TYPE csp_case_glue_ls_accU_upperPosition_enum :
(
	CSP_CASE_GLUE_LS_ACCU_UPPERPOSITION_STATUS_NOT_INITIALIZED 									:= 0,
	CSP_CASE_GLUE_LS_ACCU_UPPERPOSITION_STATUS_DISABLED 										:= 10,
	CSP_CASE_GLUE_LS_ACCU_UPPERPOSITION_STATUS_POSITION_CHECK									:= 20,
	CSP_CASE_GLUE_LS_ACCU_UPPERPOSITION_STATUS_ENABLE_REQUEST 									:= 30,
	CSP_CASE_GLUE_LS_ACCU_UPPERPOSITION_STATUS_ENABLED 											:= 40,
	CSP_CASE_GLUE_LS_ACCU_UPPERPOSITION_STATUS_ABS_MOVE_REQUEST									:= 50,
	CSP_CASE_GLUE_LS_ACCU_UPPERPOSITION_STATUS_ABS_MOVING										:= 60,
	CSP_CASE_GLUE_LS_ACCU_UPPERPOSITION_STATUS_STOP_REQUEST 									:= 70,
	CSP_CASE_GLUE_LS_ACCU_UPPERPOSITION_STATUS_DISABLE_REQUEST 									:= 80,
	CSP_CASE_GLUE_LS_ACCU_UPPERPOSITION_STATUS_DISABLING 										:= 90
) := CSP_CASE_GLUE_LS_ACCU_UPPERPOSITION_STATUS_NOT_INITIALIZED;
END_TYPE

(* stored: Version 1.1.0.1, ProductVersion 3.1.4022.18
   DUT csp_case_glue_ls_accU_upperPosition_enum: Id {6e0bb2fc-9d42-4cc0-bbab-af75d678d447} *)
